// TIA Portal V20 export
DATA_BLOCK "EQUIPMENT_DATA_SCADA_DB"   // DB201
{ S7_Optimized_Access := 'TRUE' }
// stored: AutoNumber false, MemoryReserve 100
   VAR
      PLC1_OPMODE01 { ExternalWritable := 'False'} : "EQUIPMENT_DATA_OUT_UDT";
      PLC1_OPMODE02 { ExternalWritable := 'False'} : "EQUIPMENT_DATA_OUT_UDT";
      PLC1_OPMODE03 { ExternalWritable := 'False'} : "EQUIPMENT_DATA_OUT_UDT";
      PLC1_OPMODE04 { ExternalWritable := 'False'} : "EQUIPMENT_DATA_OUT_UDT";
      PLC1_OPMODE05 { ExternalWritable := 'False'} : "EQUIPMENT_DATA_OUT_UDT";
      PLC1_OPMODE06 { ExternalWritable := 'False'} : "EQUIPMENT_DATA_OUT_UDT";
      PLC1_OPMODE01_ST010 { ExternalWritable := 'False'} : "EQUIPMENT_DATA_OUT_UDT";
      PLC1_OPMODE02_Buffer { ExternalWritable := 'False'} : "EQUIPMENT_DATA_OUT_UDT";
      PLC1_OPMODE03_Buffer { ExternalWritable := 'False'} : "EQUIPMENT_DATA_OUT_UDT";
      PLC1_OPMODE04_Buffer { ExternalWritable := 'False'} : "EQUIPMENT_DATA_OUT_UDT";
      PLC1_OPMODE05_ST020 { ExternalWritable := 'False'} : "EQUIPMENT_DATA_OUT_UDT";
      PLC1_OPMODE06_ST025 { ExternalWritable := 'False'} : "EQUIPMENT_DATA_OUT_UDT";
      PLC1_OPMODE06_ST030 { ExternalWritable := 'False'} : "EQUIPMENT_DATA_OUT_UDT";
      PLC1_OPMODE06_ST035 { ExternalWritable := 'False'} : "EQUIPMENT_DATA_OUT_UDT";
      TEST_EqtData { ExternalWritable := 'False'} : "EQUIPMENT_DATA_OUT_UDT";
   END_VAR
BEGIN
END_DATA_BLOCK
